ABB RobotStudio station: Turing_v4.rspag

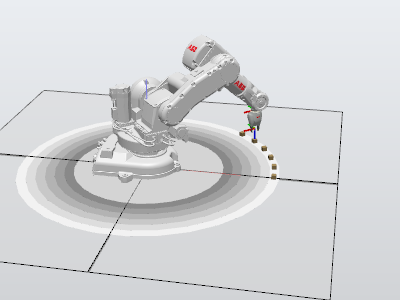
--- station ---
Station Project4 (saved by RobotStudio 24.2.10821.1)
Controller IRB140_6_81
  mechanical unit ROB_1: IRB140_6_81_C_03, 6 joints, base frame (0, 0, 0) mm
Layout (positions relative to the parent item):
  - IRB140_6_81_C_03 [mechanism, from %ABB.RobotStudio.Models.IRB140%\IRB140_6_81_C_G_03.rslib] at (0, 0, 0) mm; joint values [0.6981, 1.0743, -0.3328, 0, 0.8118, 0] (rad or m)
  - Smart_Gripper_Servo_Fingers [mechanism, from %ABB.RobotStudio.Models.SmartGripper%\ABB_Smart_Gripper_Servo_Fingers.rslib] at (511.66, 429.33, 201.88) mm, rotated rx 180 ry 1.01 rz -140 deg; joint values [0.0191] (rad or m)
  - PlaneSensor [smart component, from Components\PlaneSensor.rslib] at (513.2, 430.63, 87.7) mm, rotated rx 180 ry 1.01 rz -140 deg
      properties: Origin=[-0.0195132293626005 -0.00499999960902282 0.00895782227134504]; Axis1=[0.04 0 0]; Axis2=[1.23549883534604E-10 0.01 8.80825497109042E-11]; Tag=(none); SensedPart=(none)
    - _sensorPart_ [part], size 40 x 10 x 0 mm
  - Box_1 [part] at (-0.01, 0, -2.45) mm, size 25 x 25 x 25 mm
  - RapidVariable [smart component, from Components\RapidVariable.rslib]
      properties: DataType=bool; Controller=IRB140_6_81; Task=T_ROB1; Module=module1; Variable=plane; Value=false
  - Symbol_ring1 [part], size 1400 x 1392.3 x 0.1 mm
  - Symbol_ring2 [part], size 1300 x 1292.9 x 0.1 mm
  - Symbol_ring3 [part], size 1200 x 1193.4 x 0.1 mm
  - Symbol_ring4 [part], size 1100 x 1094 x 0.1 mm
  - Symbol_ring5 [part], size 1000 x 994.5 x 0.1 mm
  - Symbol_ring6 [part], size 900 x 895.1 x 0.1 mm
  - Base [part], size 800 x 795.6 x 0.1 mm
  - Attacher [smart component, from Components\Attacher.rslib]
      properties: Parent=Smart_Gripper_Servo_Fingers; Flange=0; Child=(none); Mount=false; Offset=[0 0 0]; Orientation=[0 0 0]
  - Detacher [smart component, from Components\Detacher.rslib]
      properties: Child=(none); KeepPosition=true
  - PoseMover [smart component, from Components\PoseMover.rslib] at (513.2, 430.63, 87.7) mm, rotated rx 180 ry 1.01 rz -140 deg
      properties: Mechanism=Smart_Gripper_Servo_Fingers; Pose=2; Duration=0
  - PoseMover_2 [smart component, from Components\PoseMover.rslib]
      properties: Mechanism=Smart_Gripper_Servo_Fingers; Pose=3; Duration=0.2
  - Box_2 [part] at (-0.01, 0, -2.45) mm, rotated rx 0 ry 0 rz 10 deg, size 25 x 25 x 25 mm
  - Box_3 [part] at (-0.01, 0, -2.45) mm, rotated rx 0 ry 0 rz 20 deg, size 25 x 25 x 25 mm
  - Box_4 [part] at (-0.01, 0, -2.45) mm, rotated rx 0 ry 0 rz 30 deg, size 25 x 25 x 25 mm
  - Box_5 [part] at (0, 0, -2.45) mm, rotated rx 0 ry 0 rz 40 deg, size 25 x 25 x 25 mm
  - Box_6 [part] at (0, 0, -2.45) mm, rotated rx 0 ry 0 rz 50 deg, size 25 x 25 x 25 mm
Attachment: Smart_Gripper_Servo_Fingers is attached to IRB140_6_81_C_03 / Link6
Attachment: PlaneSensor is attached to Smart_Gripper_Servo_Fingers / HandBase
Attachment: PoseMover is attached to Smart_Gripper_Servo_Fingers / HandBase
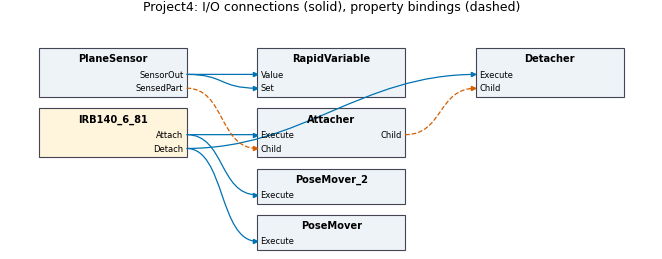
Station logic (signal -> signal, property => property):
  PlaneSensor.SensorOut -> RapidVariable.Value
  PlaneSensor.SensorOut -> RapidVariable.Set
  IRB140_6_81.Attach -> Attacher.Execute
  IRB140_6_81.Detach -> Detacher.Execute
  IRB140_6_81.Detach -> PoseMover.Execute
  IRB140_6_81.Attach -> PoseMover_2.Execute
  PlaneSensor.SensedPart => Attacher.Child
  Attacher.Child => Detacher.Child

--- Controller Data/IRB140_6_81/RAPID/TASK1/PROGMOD/CalibData.mod ---
MODULE CalibData
    PERS tooldata Servo:=[TRUE,[[0,0,114.2],[1,0,0,0]],[0.215,[8.7,12.3,49.2],[1,0,0,0],0.00021,0.00024,0.00009]];
ENDMODULE

--- Controller Data/IRB140_6_81/RAPID/TASK1/PROGMOD/Module1.mod ---
MODULE Module1
    !***********************************************************
    !
    ! Module:  Module1
    !
    ! Description:
    !   Testing code for running Turing simulators
    !
    ! Author: Mika Letonsaari
    !
    ! Version: 1.0
    !
    !***********************************************************

    ! Select the program here
    ! 1 = move pieces randomly to test it
    ! 2 = move all pieces to state 1 to initialize tape
    ! 10 = run UTM(4,6)
    VAR num program := 2;

    PERS jointtarget down{6}:= [
        [[0,68.92,-22.27,0,42.35,0], [9E9,9E9,9E9,9E9,9E9,9E9]],
        [[0,63.95,-10.59,0,35.64,0], [9E9,9E9,9E9,9E9,9E9,9E9]],
        [[0,59.56,0.48,0,28.96,0], [9E9,9E9,9E9,9E9,9E9,9E9]],
        [[0,56.07,10.18,0,22.76,0], [9E9,9E9,9E9,9E9,9E9,9E9]],
        [[0,53.14,19.57,0,16.30,0], [9E9,9E9,9E9,9E9,9E9,9E9]],
        [[0,51.01,28.28,0,9.72,0], [9E9,9E9,9E9,9E9,9E9,9E9]]
        ];
    PERS jointtarget up{6} := [
        [[0,61.55,-19.07,0,46.51,0], [9E9,9E9,9E9,9E9,9E9,9E9]],
        [[0,55.11,-5.13,0,39,0], [9E9,9E9,9E9,9E9,9E9,9E9]],
        [[0,50.59,5.04,0,33.36,0], [9E9,9E9,9E9,9E9,9E9,9E9]],
        [[0,46.51,14.67,0,27.82,0], [9E9,9E9,9E9,9E9,9E9,9E9]],
        [[0,42.80,24.01,0,22.18,0], [9E9,9E9,9E9,9E9,9E9,9E9]],
        [[0,39.78,32.41,0,16.80,0], [9E9,9E9,9E9,9E9,9E9,9E9]]
    ];
    VAR bool plane;
    VAR num angle := 0;
    VAR num q := 1;
    VAR num delay := 0.5;
    VAR num a := 0;
    VAR num stp := 10;
    VAR num dir := 1;

    PROC Main()
        SetDo Attach, 0;
        SetDo Detach, 0;
        MoveAbsJ up{1}, v100, fine, tool0;
        WaitTime delay;

        ! Program 1
        ! An example of moving pieces in random

        WHILE program = 1 DO
             GetSymbol;
             IF q = 0 THEN
                 dir := -dir;
                 q := 1;
             ELSE
                SetSymbol (1 + Trunc(Rand()/RAND_MAX*6));
            ENDIF
            IF dir > 0 THEN
                 StepForward;
            ELSE
                 StepBack;
            ENDIF
        ENDWHILE

        ! Program 2
        ! An example of moving pieces in random

        WHILE program = 2 DO
             GetSymbol;
             IF q = 0 THEN
                 EXIT;
             ELSE
                 SetSymbol (1);
             ENDIF
             StepForward;
        ENDWHILE

        ! Program 10
        ! UTM(4,6) code generated from Twine Twee file

        IF program = 10 THEN


Start:
GetSymbol;
Test q
Case 1:
    Goto q1_1;
Case 2:
    Goto q1_2;
Case 3:
    Goto q1_3;
Case 4:
    Goto q1_4;
Case 5:
    Goto q1_5;
Case 6:
    Goto q1_6;
DEFAULT :
    Goto Halt;
ENDTEST

q1:
GetSymbol;
Test q
Case 1:
    Goto q1_1;
Case 2:
    Goto q1_2;
Case 3:
    Goto q1_3;
Case 4:
    Goto q1_4;
Case 5:
    Goto q1_5;
Case 6:
    Goto q1_6;
DEFAULT :
    Goto Halt;
ENDTEST

q1_1:
SetSymbol (2);
StepBack;
Goto q2;

q1_2:
SetSymbol (3);
StepForward;
Goto q3;

q1_3:
SetSymbol (4);
StepBack;
Goto q2;

q1_4:
SetSymbol (5);
StepForward;
Goto q3;

q1_5:
SetSymbol (6);
StepBack;
Goto q2;

q1_6:
SetSymbol (1);
StepForward;
Goto q3;

q2:
GetSymbol;
Test q
Case 1:
    Goto q2_1;
Case 2:
    Goto q2_2;
Case 3:
    Goto q2_3;
Case 4:
    Goto q2_4;
Case 5:
    Goto q2_5;
Case 6:
    Goto q2_6;
DEFAULT :
    Goto Halt;
ENDTEST

q2_1:
SetSymbol (4);
StepBack;
Goto q1;

q2_2:
SetSymbol (5);
StepForward;
Goto q4;

q2_3:
SetSymbol (1);
StepBack;
Goto q1;

q2_4:
SetSymbol (2);
StepForward;
Goto q4;

q2_5:
SetSymbol (3);
StepBack;
Goto q1;

q2_6:
SetSymbol (6);
StepForward;
Goto q4;

q3:
GetSymbol;
Test q
Case 1:
    Goto q3_1;
Case 2:
    Goto q3_2;
Case 3:
    Goto q3_3;
Case 4:
    Goto q3_4;
Case 5:
    Goto q3_5;
Case 6:
    Goto q3_6;
DEFAULT :
    Goto Halt;
ENDTEST

q3_1:
SetSymbol (6);
StepBack;
Goto q1;

q3_2:
SetSymbol (3);
StepForward;
Goto q2;

q3_3:
SetSymbol (2);
StepBack;
Goto q1;

q3_4:
SetSymbol (1);
StepForward;
Goto q2;

q3_5:
SetSymbol (4);
StepBack;
Goto q1;

q3_6:
SetSymbol (5);
StepForward;
Goto q2;

q4:
GetSymbol;
Test q
Case 1:
    Goto q4_1;
Case 2:
    Goto q4_2;
Case 3:
    Goto q4_3;
Case 4:
    Goto q4_4;
Case 5:
    Goto q4_5;
Case 6:
    Goto q4_6;
DEFAULT :
    Goto Halt;
ENDTEST

q4_1:
SetSymbol (1);
StepBack;
Goto Halt;

q4_2:
SetSymbol (2);
StepForward;
Goto Halt;

q4_3:
SetSymbol (3);
StepBack;
Goto Halt;

q4_4:
SetSymbol (4);
StepForward;
Goto Halt;

q4_5:
SetSymbol (5);
StepBack;
Goto Halt;

q4_6:
SetSymbol (6);
StepForward;
Goto Halt;

Halt:

        ENDIF

    ENDPROC

    PROC StepForward()
        angle := angle + stp;
    ENDPROC

    PROC StepBack()
        angle := angle - stp;
    ENDPROC

    PROC SetSymbol(num q2)
        VAR jointtarget jt1;
        VAR jointtarget jt2;
        jt1 := up{q};
        jt1.robax.rax_1 := angle;
        MoveAbsJ jt1, v100, fine, tool0;
        WaitTime delay;
        jt2 := down{q};
        jt2.robax.rax_1 := angle;
        MoveAbsJ jt2, v100, fine, tool0;
        SetDo Attach, 1;
        WaitTime delay;
        SetDo Attach, 0;
        MoveAbsJ jt1, v100, fine, tool0;
        WaitTime delay;

        jt1 := up{q2};
        jt1.robax.rax_1 := angle;
        MoveAbsJ jt1, v100, fine, tool0;
        WaitTime delay;
        jt2 := down{q2};
        jt2.robax.rax_1 := angle;
        MoveAbsJ jt2, v100, fine, tool0;
        SetDo Detach, 1;
        WaitTime delay;
        SetDo Detach, 0;
        MoveAbsJ jt1, v100, fine, tool0;
        WaitTime delay;

    ENDPROC

    PROC GetSymbol ()
        VAR jointtarget jt1;
        VAR jointtarget jt2;
        plane := FALSE;
        q := 1;
        WHILE q < 7 DO
            jt1 := up{q};
            jt1.robax.rax_1 := angle;
            MoveAbsJ jt1, v100, fine, tool0;
            WaitTime delay;
            jt2 := down{q};
            jt2.robax.rax_1 := angle;
            MoveAbsJ jt2, v100, fine, tool0;
            WaitTime delay;
            IF plane THEN
                WHILE angle < 0 DO
                    WaitTime delay;
                ENDWHILE
                MoveAbsJ jt1, v100, fine, tool0;
                WaitTime delay;
                RETURN;
            ENDIF
            MoveAbsJ jt1, v100, fine, tool0;
            WaitTime delay;
            q := q + 1;
        ENDWHILE
        q := 0;
    ENDPROC

ENDMODULE

--- Controller Data/IRB140_6_81/SYSPAR/EIO.cfg ---
EIO:CFG_1.0:6:1::
#
EIO_SIGNAL:

      -Name "Attach" -SignalType "DO"

      -Name "Detach" -SignalType "DO"
